// TIA Portal V17 export
// export: Created 2023-02-25T14:37:14.8109943Z, ExportSetting WithDefaults, DisplayName Totally Integrated Automation Portal, DisplayVersion V17, DisplayName TIA Portal Openness, DisplayVersion V17, DisplayName TIA Portal Version Control Interface, DisplayVersion V17, DisplayName TIA Portal Test Suite Advanced, DisplayVersion V17, DisplayName STEP 7 Professional, DisplayVersion V17, DisplayName SIMATIC Energy Suite, DisplayVersion V17, DisplayName STEP 7 Safety, DisplayVersion V17, DisplayName WinCC Professional, DisplayVersion V17
VAR_GLOBAL   // PLC tag table "Output"
   O_W AT %Q0.0 : Bool;
   O_SendLeft AT %Q0.1 : Bool;
   O_SendRight AT %Q0.2 : Bool;
   O_SendForward AT %Q0.3 : Bool;
   O_StartLight AT %Q0.4 : Bool;
   O_ResetLight AT %Q0.5 : Bool;
   O_StopLight AT %Q0.6 : Bool;
   O_ColumnRed AT %Q0.7 : Bool;
   O_ColumnGreen AT %Q1.0 : Bool;
   O_ColumnYellow AT %Q1.1 : Bool;
   O_C1_light AT %Q1.2 : Bool;
   O_C3_light AT %Q1.4 : Bool;
   O_C4_light AT %Q1.5 : Bool;
   O_C5_light AT %Q1.6 : Bool;
   O_SendLeft_light AT %Q1.7 : Bool;
   O_SendForward_light AT %Q2.0 : Bool;
   O_SendRight_light AT %Q2.1 : Bool;
   O_ResetCount_light AT %Q2.2 : Bool;
   O_AlarmSiren AT %Q2.3 : Bool;
   O_C2_light AT %Q1.3 : Bool;
   O_LeftCount AT %QD30 : DInt;
   O_ForwardCount AT %QD34 : DInt;
   O_RightCOunt AT %QD38 : DInt;
   O_Weight AT %QD42 : Real;
   O_C1 AT %QD46 : DInt;
   O_C2 AT %QD50 : DInt;
   O_C3 AT %QD54 : DInt;
   O_C4 AT %QD58 : DInt;
END_VAR
